(* IEC 61131-3 sources: com.logicals.lc3.webinar/usRTS_RPMControl_iSOC/src_FB_LIB_SAFE/Convert/REAL, 2 files *)

(* ---- wREAL_TO_LREAL.iecst ---- *)
NAMESPACE logicals.web.standard
NAMESPACE convert

/*
 * Function block wrapper for IEC 61131-3 TO_LREAL<br>
 * IN =  input value (REAL)<br>
 * OUT = IN (LREAL)<br>
 */
FUNCTION_BLOCK wREAL_TO_LREAL
	{ vNameAlignment:="center"; altName:="REAL_TO_LREAL"; bgColor:="Orange"; width:=140; hideIONames; }
	VAR_INPUT
		IN : REAL;
	END_VAR
	VAR_OUTPUT
		OUT: LREAL;
	END_VAR

	OUT := TO_LREAL(IN:=IN, ENO=>ENO);
END_FUNCTION_BLOCK

END_NAMESPACE
END_NAMESPACE

(* ---- wTRUNC_REAL_TO_LINT.iecst ---- *)
NAMESPACE logicals.web.standard
NAMESPACE convert

/*
 * Function block wrapper for IEC 61131-3 TO_LINT<br>
 * IN =  input value (REAL)<br>
 * OUT = IN (LINT)<br>
 */
FUNCTION_BLOCK wTRUNC_REAL_TO_LINT
	{ vNameAlignment:="center"; altName:="TRUNC_REAL_TO_LINT"; bgColor:="LightPink"; width:=180; hideIONames; }
	VAR_INPUT
		IN : REAL;
	END_VAR
	VAR_OUTPUT
		OUT: LINT;
	END_VAR

	OUT := TO_LINT(IN:=IN, ENO=>ENO);
END_FUNCTION_BLOCK

END_NAMESPACE
END_NAMESPACE
